FUNCTION_BLOCK ChamberGaugeViewModule
VAR_INPUT
	inputValue:DINT;// 输入值
	gaugeType:INT;// 类型，1：AIM；2：PSG
	calValueH:REAL;// 计算值上限
	calValueL:REAL;// 计算值下限
	moduleValueH:REAL;// 模块上限
	moduleValueL:REAL;// 模块下限
	alrmmaxValue:REAL;// 警告上限
	alrmminValue:REAL;// 警告下限
	condition:BOOL;// 显示条件
	initString:STRING:='-----';// 初始显示字符串：*****
END_VAR
VAR_OUTPUT
	outputValue:REAL;
	outputValue1:REAL;
	outputValue_String:STRING;
	error:BOOL;
END_VAR
VAR
	factor:REAL;// 转换因子
	temp:REAL;
	test:REAL;
	tT:TON;
END_VAR

IF ((moduleValueH-moduleValueL)>0.0) THEN
	factor:=(calValueH-calValueL)/(moduleValueH-moduleValueL);
	temp:=factor*DINT_TO_REAL(inputValue);
	outputValue:=temp*((alrmmaxValue-alrmminValue)/(19-4));
//	IF outputValue<100000 THEN
//		outputValue_String:=REAL_TO_STRING(outputValue-1100);
//		outputValue1:=(outputValue-1100);
//	ELSE
//		outputValue_String:=REAL_TO_STRING(outputValue);
//		outputValue1:=(outputValue);
//	END_IF
	IF outputValue-1100<1 THEN
		outputValue:=1112.4;
	END_IF
	outputValue_String:=REAL_TO_STRING(outputValue-1100);
	outputValue1:=(outputValue-1100);
	tT(IN:=NOT (( outputValue>alrmminValue) AND inputValue>10),PT:=T#2S);
	IF tT.Q THEN
		error:=TRUE;
	ELSE
		error:=FALSE;
	END_IF
	
	IF condition THEN
		;
	ELSE
		outputValue_String:=initString;
	END_IF
END_IF

END_FUNCTION_BLOCK

(* stored: Version 1.1.0.1, ProductVersion 3.1.4024.12
   POU ChamberGaugeViewModule: Id {373cbe64-6a33-4413-9035-9fef5e8ee2fe}, SpecialFunc None *)
